REGION Network 98: Step[822] : Side Tape Attachment Y-Axis Remain Attach Right Position
   RUNG wire#powerrail
      { S7_Templates := "SrcType := DInt" } EQ_Contact(in1 := "Unit1.Em4.ControlNodes".sideTapeAttachment.sequence.status.currentStep, in2 := #JOB_8_STEP_22)
      Contact( "Unit1.Em4.ControlNodes".sideTapeAttachment.sequence.status.seqActive )
      wire#w1
      I_Contact( "Unit1.Em4.ControlNodes".cm.softcam.sideTapeAttachmentAxisY.pos08_remainAttachRight.inPos )
      Coil( "Unit1.Em4.ControlNodes".sideTapeAttachment."step".action1[822] )
   END_RUNG
   RUNG wire#w1
      Contact( "JB_Temp".Test_sig_4[2, 8, 7] )
      Contact( "Unit1.Em4.ControlNodes".cm.softcam.sideTapeAttachmentAxisY.pos08_remainAttachRight.inPos )
      Coil( "Unit1.Em4.ControlNodes".sideTapeAttachment."step".transition1[822] )
   END_RUNG
   RUNG wire#w1
      Contact( "Unit1.Em4.ControlNodes".sideTapeAttachment."step".transition1[822] )
      { S7_Templates := "time_type := Time" } #statTonTime[822].TON(pt := T#500ms, et =>)
      Move(in := #JOB_8_STEP_23, out1 => "Unit1.Em4.ControlNodes".sideTapeAttachment.sequence.status.nextStep)
   END_RUNG
   // the same network as SCL:
   #_w1 := ("Unit1.Em4.ControlNodes".sideTapeAttachment.sequence.status.currentStep = #JOB_8_STEP_22) AND "Unit1.Em4.ControlNodes".sideTapeAttachment.sequence.status.seqActive;
   "Unit1.Em4.ControlNodes".sideTapeAttachment."step".action1[822] := #_w1 AND NOT "Unit1.Em4.ControlNodes".cm.softcam.sideTapeAttachmentAxisY.pos08_remainAttachRight.inPos;
   "Unit1.Em4.ControlNodes".sideTapeAttachment."step".transition1[822] := #_w1 AND "JB_Temp".Test_sig_4[2, 8, 7] AND "Unit1.Em4.ControlNodes".cm.softcam.sideTapeAttachmentAxisY.pos08_remainAttachRight.inPos;
   #statTonTime[822].TON(IN := #_w1 AND "Unit1.Em4.ControlNodes".sideTapeAttachment."step".transition1[822],
                         PT := T#500ms);
   IF #statTonTime[822].Q THEN
       "Unit1.Em4.ControlNodes".sideTapeAttachment.sequence.status.nextStep := #JOB_8_STEP_23;
   END_IF;
END_REGION

REGION Network 99: Step[823] : Side Tape Attachment Right Vaccum Off
   RUNG wire#powerrail
      { S7_Templates := "SrcType := DInt" } EQ_Contact(in1 := "Unit1.Em4.ControlNodes".sideTapeAttachment.sequence.status.currentStep, in2 := #JOB_8_STEP_23)
      Contact( "Unit1.Em4.ControlNodes".sideTapeAttachment.sequence.status.seqActive )
      wire#w1
      I_Contact( "Unit1.Em4.ControlNodes".cmSideTapeAttachment2TopVaccumOffOn.monitoring.inHomePos )
      wire#w2
      Coil( "Unit1.Em4.ControlNodes".sideTapeAttachment."step".action1[823] )
   END_RUNG
   RUNG wire#w1
      I_Contact( "Unit1.Em4.ControlNodes".cmSideTapeAttachment2BtmVaccumOffOn.monitoring.inHomePos )
   END_RUNG wire#w2
   RUNG wire#w1
      Contact( "JB_Temp".Test_sig_4[2, 8, 8] )
      Contact( "Unit1.Em4.ControlNodes".cmSideTapeAttachment2TopVaccumOffOn.monitoring.inHomePos )
      Contact( "Unit1.Em4.ControlNodes".cmSideTapeAttachment2BtmVaccumOffOn.monitoring.inHomePos )
      Coil( "Unit1.Em4.ControlNodes".sideTapeAttachment."step".transition1[823] )
   END_RUNG
   RUNG wire#w1
      Contact( "Unit1.Em4.ControlNodes".sideTapeAttachment."step".transition1[823] )
      { S7_Templates := "time_type := Time" } #statTonTime[823].TON(pt := T#500ms, et =>)
      Move(in := #JOB_8_STEP_24, out1 => "Unit1.Em4.ControlNodes".sideTapeAttachment.sequence.status.nextStep)
   END_RUNG
   // the same network as SCL:
   #_w1 := ("Unit1.Em4.ControlNodes".sideTapeAttachment.sequence.status.currentStep = #JOB_8_STEP_23) AND "Unit1.Em4.ControlNodes".sideTapeAttachment.sequence.status.seqActive;
   "Unit1.Em4.ControlNodes".sideTapeAttachment."step".action1[823] := #_w1 AND (NOT "Unit1.Em4.ControlNodes".cmSideTapeAttachment2TopVaccumOffOn.monitoring.inHomePos OR NOT "Unit1.Em4.ControlNodes".cmSideTapeAttachment2BtmVaccumOffOn.monitoring.inHomePos);
   "Unit1.Em4.ControlNodes".sideTapeAttachment."step".transition1[823] := #_w1 AND "JB_Temp".Test_sig_4[2, 8, 8] AND "Unit1.Em4.ControlNodes".cmSideTapeAttachment2TopVaccumOffOn.monitoring.inHomePos AND "Unit1.Em4.ControlNodes".cmSideTapeAttachment2BtmVaccumOffOn.monitoring.inHomePos;
   #statTonTime[823].TON(IN := #_w1 AND "Unit1.Em4.ControlNodes".sideTapeAttachment."step".transition1[823],
                         PT := T#500ms);
   IF #statTonTime[823].Q THEN
       "Unit1.Em4.ControlNodes".sideTapeAttachment.sequence.status.nextStep := #JOB_8_STEP_24;
   END_IF;
END_REGION

REGION Network 100: Step[824] : Side Tape Attachment Y-Axis Wait Pos
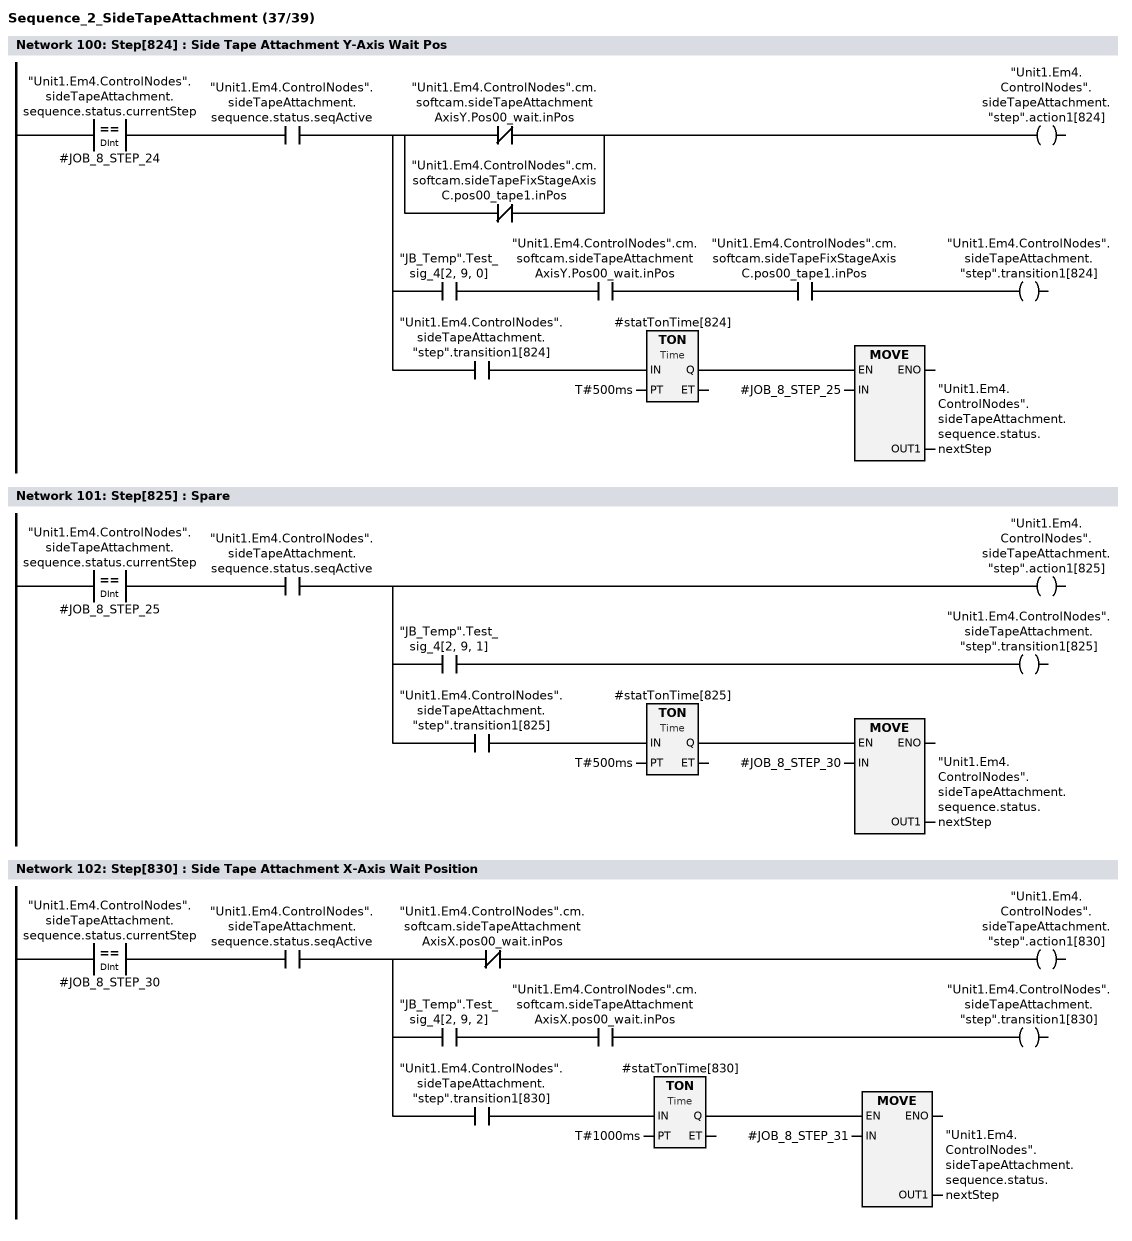
   RUNG wire#powerrail
      { S7_Templates := "SrcType := DInt" } EQ_Contact(in1 := "Unit1.Em4.ControlNodes".sideTapeAttachment.sequence.status.currentStep, in2 := #JOB_8_STEP_24)
      Contact( "Unit1.Em4.ControlNodes".sideTapeAttachment.sequence.status.seqActive )
      wire#w1
      I_Contact( "Unit1.Em4.ControlNodes".cm.softcam.sideTapeAttachmentAxisY.Pos00_wait.inPos )
      wire#w2
      Coil( "Unit1.Em4.ControlNodes".sideTapeAttachment."step".action1[824] )
   END_RUNG
   RUNG wire#w1
      I_Contact( "Unit1.Em4.ControlNodes".cm.softcam.sideTapeFixStageAxisC.pos00_tape1.inPos )
   END_RUNG wire#w2
   RUNG wire#w1
      Contact( "JB_Temp".Test_sig_4[2, 9, 0] )
      Contact( "Unit1.Em4.ControlNodes".cm.softcam.sideTapeAttachmentAxisY.Pos00_wait.inPos )
      Contact( "Unit1.Em4.ControlNodes".cm.softcam.sideTapeFixStageAxisC.pos00_tape1.inPos )
      Coil( "Unit1.Em4.ControlNodes".sideTapeAttachment."step".transition1[824] )
   END_RUNG
   RUNG wire#w1
      Contact( "Unit1.Em4.ControlNodes".sideTapeAttachment."step".transition1[824] )
      { S7_Templates := "time_type := Time" } #statTonTime[824].TON(pt := T#500ms, et =>)
      Move(in := #JOB_8_STEP_25, out1 => "Unit1.Em4.ControlNodes".sideTapeAttachment.sequence.status.nextStep)
   END_RUNG
   // the same network as SCL:
   #_w1 := ("Unit1.Em4.ControlNodes".sideTapeAttachment.sequence.status.currentStep = #JOB_8_STEP_24) AND "Unit1.Em4.ControlNodes".sideTapeAttachment.sequence.status.seqActive;
   "Unit1.Em4.ControlNodes".sideTapeAttachment."step".action1[824] := #_w1 AND (NOT "Unit1.Em4.ControlNodes".cm.softcam.sideTapeAttachmentAxisY.Pos00_wait.inPos OR NOT "Unit1.Em4.ControlNodes".cm.softcam.sideTapeFixStageAxisC.pos00_tape1.inPos);
   "Unit1.Em4.ControlNodes".sideTapeAttachment."step".transition1[824] := #_w1 AND "JB_Temp".Test_sig_4[2, 9, 0] AND "Unit1.Em4.ControlNodes".cm.softcam.sideTapeAttachmentAxisY.Pos00_wait.inPos AND "Unit1.Em4.ControlNodes".cm.softcam.sideTapeFixStageAxisC.pos00_tape1.inPos;
   #statTonTime[824].TON(IN := #_w1 AND "Unit1.Em4.ControlNodes".sideTapeAttachment."step".transition1[824],
                         PT := T#500ms);
   IF #statTonTime[824].Q THEN
       "Unit1.Em4.ControlNodes".sideTapeAttachment.sequence.status.nextStep := #JOB_8_STEP_25;
   END_IF;
END_REGION

REGION Network 101: Step[825] : Spare
   RUNG wire#powerrail
      { S7_Templates := "SrcType := DInt" } EQ_Contact(in1 := "Unit1.Em4.ControlNodes".sideTapeAttachment.sequence.status.currentStep, in2 := #JOB_8_STEP_25)
      Contact( "Unit1.Em4.ControlNodes".sideTapeAttachment.sequence.status.seqActive )
      wire#w1
      Coil( "Unit1.Em4.ControlNodes".sideTapeAttachment."step".action1[825] )
   END_RUNG
   RUNG wire#w1
      Contact( "JB_Temp".Test_sig_4[2, 9, 1] )
      Coil( "Unit1.Em4.ControlNodes".sideTapeAttachment."step".transition1[825] )
   END_RUNG
   RUNG wire#w1
      Contact( "Unit1.Em4.ControlNodes".sideTapeAttachment."step".transition1[825] )
      { S7_Templates := "time_type := Time" } #statTonTime[825].TON(pt := T#500ms, et =>)
      Move(in := #JOB_8_STEP_30, out1 => "Unit1.Em4.ControlNodes".sideTapeAttachment.sequence.status.nextStep)
   END_RUNG
   // the same network as SCL:
   "Unit1.Em4.ControlNodes".sideTapeAttachment."step".action1[825] := ("Unit1.Em4.ControlNodes".sideTapeAttachment.sequence.status.currentStep = #JOB_8_STEP_25) AND "Unit1.Em4.ControlNodes".sideTapeAttachment.sequence.status.seqActive;
   "Unit1.Em4.ControlNodes".sideTapeAttachment."step".transition1[825] := ("Unit1.Em4.ControlNodes".sideTapeAttachment.sequence.status.currentStep = #JOB_8_STEP_25) AND "Unit1.Em4.ControlNodes".sideTapeAttachment.sequence.status.seqActive AND "JB_Temp".Test_sig_4[2, 9, 1];
   #statTonTime[825].TON(IN := ("Unit1.Em4.ControlNodes".sideTapeAttachment.sequence.status.currentStep = #JOB_8_STEP_25) AND "Unit1.Em4.ControlNodes".sideTapeAttachment.sequence.status.seqActive AND "Unit1.Em4.ControlNodes".sideTapeAttachment."step".transition1[825],
                         PT := T#500ms);
   IF #statTonTime[825].Q THEN
       "Unit1.Em4.ControlNodes".sideTapeAttachment.sequence.status.nextStep := #JOB_8_STEP_30;
   END_IF;
END_REGION

REGION Network 102: Step[830] : Side Tape Attachment X-Axis Wait Position
   RUNG wire#powerrail
      { S7_Templates := "SrcType := DInt" } EQ_Contact(in1 := "Unit1.Em4.ControlNodes".sideTapeAttachment.sequence.status.currentStep, in2 := #JOB_8_STEP_30)
      Contact( "Unit1.Em4.ControlNodes".sideTapeAttachment.sequence.status.seqActive )
      wire#w1
      I_Contact( "Unit1.Em4.ControlNodes".cm.softcam.sideTapeAttachmentAxisX.pos00_wait.inPos )
      Coil( "Unit1.Em4.ControlNodes".sideTapeAttachment."step".action1[830] )
   END_RUNG
   RUNG wire#w1
      Contact( "JB_Temp".Test_sig_4[2, 9, 2] )
      Contact( "Unit1.Em4.ControlNodes".cm.softcam.sideTapeAttachmentAxisX.pos00_wait.inPos )
      Coil( "Unit1.Em4.ControlNodes".sideTapeAttachment."step".transition1[830] )
   END_RUNG
   RUNG wire#w1
      Contact( "Unit1.Em4.ControlNodes".sideTapeAttachment."step".transition1[830] )
      { S7_Templates := "time_type := Time" } #statTonTime[830].TON(pt := T#1000ms, et =>)
      Move(in := #JOB_8_STEP_31, out1 => "Unit1.Em4.ControlNodes".sideTapeAttachment.sequence.status.nextStep)
   END_RUNG
   // the same network as SCL:
   #_w1 := ("Unit1.Em4.ControlNodes".sideTapeAttachment.sequence.status.currentStep = #JOB_8_STEP_30) AND "Unit1.Em4.ControlNodes".sideTapeAttachment.sequence.status.seqActive;
   "Unit1.Em4.ControlNodes".sideTapeAttachment."step".action1[830] := #_w1 AND NOT "Unit1.Em4.ControlNodes".cm.softcam.sideTapeAttachmentAxisX.pos00_wait.inPos;
   "Unit1.Em4.ControlNodes".sideTapeAttachment."step".transition1[830] := #_w1 AND "JB_Temp".Test_sig_4[2, 9, 2] AND "Unit1.Em4.ControlNodes".cm.softcam.sideTapeAttachmentAxisX.pos00_wait.inPos;
   #statTonTime[830].TON(IN := #_w1 AND "Unit1.Em4.ControlNodes".sideTapeAttachment."step".transition1[830],
                         PT := T#1000ms);
   IF #statTonTime[830].Q THEN
       "Unit1.Em4.ControlNodes".sideTapeAttachment.sequence.status.nextStep := #JOB_8_STEP_31;
   END_IF;
END_REGION

REGION Network 103: Step[831] : Job[1] Step End
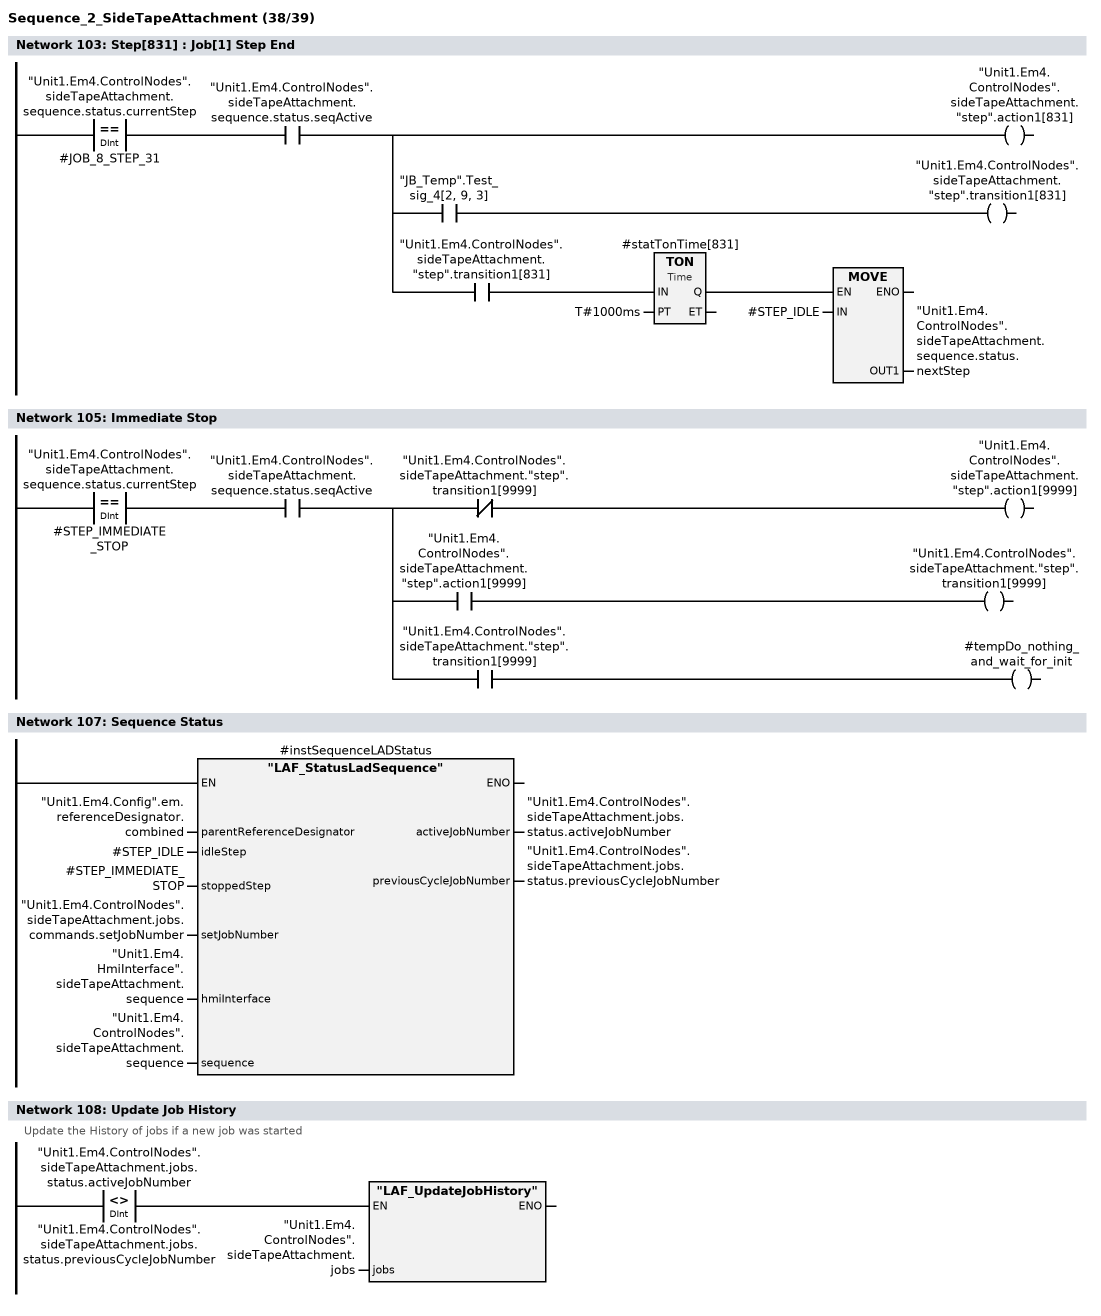
   RUNG wire#powerrail
      { S7_Templates := "SrcType := DInt" } EQ_Contact(in1 := "Unit1.Em4.ControlNodes".sideTapeAttachment.sequence.status.currentStep, in2 := #JOB_8_STEP_31)
      Contact( "Unit1.Em4.ControlNodes".sideTapeAttachment.sequence.status.seqActive )
      wire#w1
      Coil( "Unit1.Em4.ControlNodes".sideTapeAttachment."step".action1[831] )
   END_RUNG
   RUNG wire#w1
      Contact( "JB_Temp".Test_sig_4[2, 9, 3] )
      Coil( "Unit1.Em4.ControlNodes".sideTapeAttachment."step".transition1[831] )
   END_RUNG
   RUNG wire#w1
      Contact( "Unit1.Em4.ControlNodes".sideTapeAttachment."step".transition1[831] )
      { S7_Templates := "time_type := Time" } #statTonTime[831].TON(pt := T#1000ms, et =>)
      Move(in := #STEP_IDLE, out1 => "Unit1.Em4.ControlNodes".sideTapeAttachment.sequence.status.nextStep)
   END_RUNG
   // the same network as SCL:
   "Unit1.Em4.ControlNodes".sideTapeAttachment."step".action1[831] := ("Unit1.Em4.ControlNodes".sideTapeAttachment.sequence.status.currentStep = #JOB_8_STEP_31) AND "Unit1.Em4.ControlNodes".sideTapeAttachment.sequence.status.seqActive;
   "Unit1.Em4.ControlNodes".sideTapeAttachment."step".transition1[831] := ("Unit1.Em4.ControlNodes".sideTapeAttachment.sequence.status.currentStep = #JOB_8_STEP_31) AND "Unit1.Em4.ControlNodes".sideTapeAttachment.sequence.status.seqActive AND "JB_Temp".Test_sig_4[2, 9, 3];
   #statTonTime[831].TON(IN := ("Unit1.Em4.ControlNodes".sideTapeAttachment.sequence.status.currentStep = #JOB_8_STEP_31) AND "Unit1.Em4.ControlNodes".sideTapeAttachment.sequence.status.seqActive AND "Unit1.Em4.ControlNodes".sideTapeAttachment."step".transition1[831],
                         PT := T#1000ms);
   IF #statTonTime[831].Q THEN
       "Unit1.Em4.ControlNodes".sideTapeAttachment.sequence.status.nextStep := #STEP_IDLE;
   END_IF;
END_REGION

REGION Network 104: *************** IMMEDIATE STOP ****************
END_REGION

REGION Network 105: Immediate Stop
   RUNG wire#powerrail
      { S7_Templates := "SrcType := DInt" } EQ_Contact(in1 := "Unit1.Em4.ControlNodes".sideTapeAttachment.sequence.status.currentStep, in2 := #STEP_IMMEDIATE_STOP)
      Contact( "Unit1.Em4.ControlNodes".sideTapeAttachment.sequence.status.seqActive )
      wire#w1
      I_Contact( "Unit1.Em4.ControlNodes".sideTapeAttachment."step".transition1[9999] )
      Coil( "Unit1.Em4.ControlNodes".sideTapeAttachment."step".action1[9999] )
   END_RUNG
   RUNG wire#w1
      Contact( "Unit1.Em4.ControlNodes".sideTapeAttachment."step".action1[9999] )
      Coil( "Unit1.Em4.ControlNodes".sideTapeAttachment."step".transition1[9999] )
   END_RUNG
   RUNG wire#w1
      Contact( "Unit1.Em4.ControlNodes".sideTapeAttachment."step".transition1[9999] )
      Coil( #tempDo_nothing_and_wait_for_init )
   END_RUNG
   // the same network as SCL:
   #_w1 := ("Unit1.Em4.ControlNodes".sideTapeAttachment.sequence.status.currentStep = #STEP_IMMEDIATE_STOP) AND "Unit1.Em4.ControlNodes".sideTapeAttachment.sequence.status.seqActive;
   "Unit1.Em4.ControlNodes".sideTapeAttachment."step".action1[9999] := #_w1 AND NOT "Unit1.Em4.ControlNodes".sideTapeAttachment."step".transition1[9999];
   "Unit1.Em4.ControlNodes".sideTapeAttachment."step".transition1[9999] := #_w1 AND "Unit1.Em4.ControlNodes".sideTapeAttachment."step".action1[9999];
   #tempDo_nothing_and_wait_for_init := #_w1 AND "Unit1.Em4.ControlNodes".sideTapeAttachment."step".transition1[9999];
END_REGION

REGION Network 106: *************** STATUS **********************
END_REGION

REGION Network 107: Sequence Status
   RUNG wire#powerrail
      #instSequenceLADStatus(parentReferenceDesignator := "Unit1.Em4.Config".em.referenceDesignator.combined, idleStep := #STEP_IDLE, stoppedStep := #STEP_IMMEDIATE_STOP, setJobNumber := "Unit1.Em4.ControlNodes".sideTapeAttachment.jobs.commands.setJobNumber, hmiInterface := "Unit1.Em4.HmiInterface".sideTapeAttachment.sequence, sequence := "Unit1.Em4.ControlNodes".sideTapeAttachment.sequence, activeJobNumber => "Unit1.Em4.ControlNodes".sideTapeAttachment.jobs.status.activeJobNumber, previousCycleJobNumber => "Unit1.Em4.ControlNodes".sideTapeAttachment.jobs.status.previousCycleJobNumber)
   END_RUNG
   // the same network as SCL:
   #instSequenceLADStatus(parentReferenceDesignator := "Unit1.Em4.Config".em.referenceDesignator.combined,   // "LAF_StatusLadSequence"
                          idleStep := #STEP_IDLE,
                          stoppedStep := #STEP_IMMEDIATE_STOP,
                          setJobNumber := "Unit1.Em4.ControlNodes".sideTapeAttachment.jobs.commands.setJobNumber,
                          hmiInterface := "Unit1.Em4.HmiInterface".sideTapeAttachment.sequence,
                          sequence := "Unit1.Em4.ControlNodes".sideTapeAttachment.sequence,
                          activeJobNumber => "Unit1.Em4.ControlNodes".sideTapeAttachment.jobs.status.activeJobNumber,
                          previousCycleJobNumber => "Unit1.Em4.ControlNodes".sideTapeAttachment.jobs.status.previousCycleJobNumber);
END_REGION

REGION Network 108: Update Job History
   // Update the History of jobs if a new job was started
   RUNG wire#powerrail
      { S7_Templates := "SrcType := DInt" } NE_Contact(in1 := "Unit1.Em4.ControlNodes".sideTapeAttachment.jobs.status.activeJobNumber, in2 := "Unit1.Em4.ControlNodes".sideTapeAttachment.jobs.status.previousCycleJobNumber)
      "LAF_UpdateJobHistory"(jobs := "Unit1.Em4.ControlNodes".sideTapeAttachment.jobs)
   END_RUNG
   // the same network as SCL:
   IF "Unit1.Em4.ControlNodes".sideTapeAttachment.jobs.status.activeJobNumber <> "Unit1.Em4.ControlNodes".sideTapeAttachment.jobs.status.previousCycleJobNumber THEN
       "LAF_UpdateJobHistory"(jobs := "Unit1.Em4.ControlNodes".sideTapeAttachment.jobs);
   END_IF;
END_REGION

REGION Network 109: Output steps as String
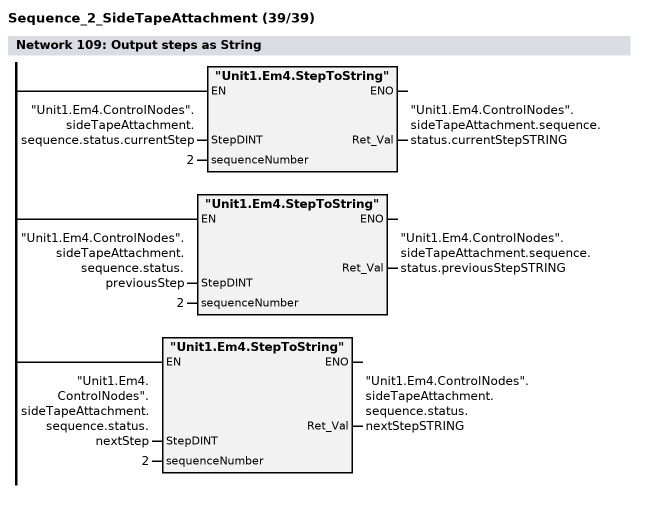
   RUNG wire#powerrail
      "Unit1.Em4.StepToString"(StepDINT := "Unit1.Em4.ControlNodes".sideTapeAttachment.sequence.status.currentStep, sequenceNumber := 2, Ret_Val => "Unit1.Em4.ControlNodes".sideTapeAttachment.sequence.status.currentStepSTRING)
   END_RUNG
   RUNG wire#powerrail
      "Unit1.Em4.StepToString"(StepDINT := "Unit1.Em4.ControlNodes".sideTapeAttachment.sequence.status.previousStep, sequenceNumber := 2, Ret_Val => "Unit1.Em4.ControlNodes".sideTapeAttachment.sequence.status.previousStepSTRING)
   END_RUNG
   RUNG wire#powerrail
      "Unit1.Em4.StepToString"(StepDINT := "Unit1.Em4.ControlNodes".sideTapeAttachment.sequence.status.nextStep, sequenceNumber := 2, Ret_Val => "Unit1.Em4.ControlNodes".sideTapeAttachment.sequence.status.nextStepSTRING)
   END_RUNG
   // the same network as SCL:
   "Unit1.Em4.ControlNodes".sideTapeAttachment.sequence.status.currentStepSTRING := "Unit1.Em4.StepToString"(StepDINT := "Unit1.Em4.ControlNodes".sideTapeAttachment.sequence.status.currentStep,
                           sequenceNumber := 2);
   "Unit1.Em4.ControlNodes".sideTapeAttachment.sequence.status.previousStepSTRING := "Unit1.Em4.StepToString"(StepDINT := "Unit1.Em4.ControlNodes".sideTapeAttachment.sequence.status.previousStep,
                           sequenceNumber := 2);
   "Unit1.Em4.ControlNodes".sideTapeAttachment.sequence.status.nextStepSTRING := "Unit1.Em4.StepToString"(StepDINT := "Unit1.Em4.ControlNodes".sideTapeAttachment.sequence.status.nextStep,
                           sequenceNumber := 2);
END_REGION
END_FUNCTION_BLOCK
